// Brief: Master Arm Initialization
FUNCTION_BLOCK PUBLIC FB_ArmReady EXTENDS FB_MasterArmCtrlBase
VAR_INPUT
END_VAR
VAR_OUTPUT
END_VAR
VAR
END_VAR

END_FUNCTION_BLOCK

(* stored: Version 1.1.0.1, ProductVersion 3.1.4024.12
   POU FB_ArmReady: Id {b4863c0c-c549-4967-ab29-6a1152ef3cd8}, SpecialFunc None *)
